// TIA Portal V16 export
// export: Created 2022-03-28T07:44:06.0907199Z, ExportSetting WithDefaults, DisplayName Totally Integrated Automation Portal, DisplayVersion V16 Update 5, DisplayName TIA Portal Version Control Interface, DisplayVersion V16 Update 2, DisplayName TIA Portal Openness, DisplayVersion V16 Update 5, DisplayName STEP 7 Professional, DisplayVersion V16 Update 5, DisplayName STEP 7 Safety, DisplayVersion V16, DisplayName WinCC Professional, DisplayVersion V16 Update 5
ORGANIZATION_BLOCK "Main"   // OB1, LAD, ProgramCycle
TITLE = "Main Program Sweep (Cycle)"
{ S7_Optimized_Access := 'TRUE' }
VERSION : 0.1
// stored: AutoNumber true, IsIECCheckEnabled false, SetENOAutomatically false
   VAR_INPUT
      Initial_Call : Bool;   // Initial call of this OB
      Remanence : Bool;   // =True, if remanent data are available
   END_VAR
BEGIN

REGION Network 1
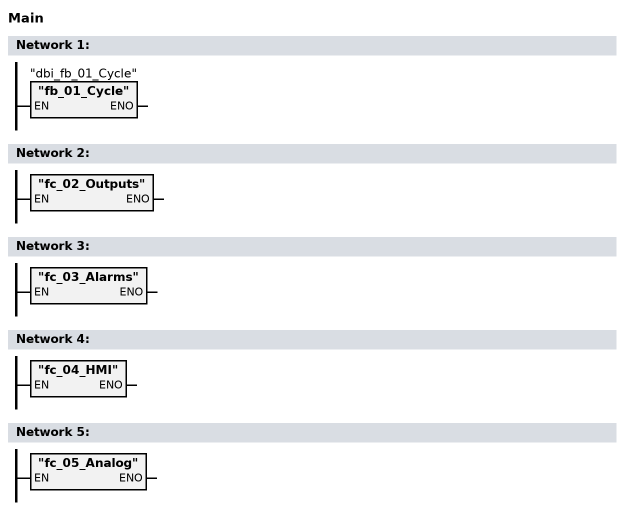
   RUNG wire#powerrail
      "dbi_fb_01_Cycle"()
   END_RUNG
   // the same network as SCL:
   "dbi_fb_01_Cycle"();   // "fb_01_Cycle"
END_REGION

REGION Network 2
   RUNG wire#powerrail
      "fc_02_Outputs"()
   END_RUNG
   // the same network as SCL:
   "fc_02_Outputs"();
END_REGION

REGION Network 3
   RUNG wire#powerrail
      "fc_03_Alarms"()
   END_RUNG
   // the same network as SCL:
   "fc_03_Alarms"();
END_REGION

REGION Network 4
   RUNG wire#powerrail
      "fc_04_HMI"()
   END_RUNG
   // the same network as SCL:
   "fc_04_HMI"();
END_REGION

REGION Network 5
   RUNG wire#powerrail
      "fc_05_Analog"()
   END_RUNG
   // the same network as SCL:
   "fc_05_Analog"();
END_REGION
END_ORGANIZATION_BLOCK
